// TIA Portal V20 export
DATA_BLOCK "BK05"   // DB194
// stored: MemoryReserve 100
   VAR
      "X10-1 SPARE" : Bool;
      "X11-1 SPARE" : Bool;
      "X12-1 COMPENSATOR LIMIT SENSOR(-)" : Bool;
      "X13-1 COMPENSATOR LIMIT SENSOR(+)" : Bool;
      "X14-1 FEEDER CYLINDER UP" : Bool;
      "X15-1 VISION PUSHER SUPPORT UP" : Bool;
      "X16-1 ELECTRODE NG BOX LOCK CYLINDER DOWN" : Bool;
      "X17-1 UNWINDER DANCER SAFETY PIN IDLE POSITION" : Bool;
      "X10-2 SPARE" : Bool;
      "X11-2 SPARE" : Bool;
      "X12-2 COMPENSATOR HOMING SENSOR" : Bool;
      "X13-2 COMPENSATOR SAFETY PIN IDLE POSITION" : Bool;
      "X14-2 FEEDER CYLINDER DOWN" : Bool;
      "X15-2 VISION PUSHER SUPPORT DOWN" : Bool;
      "X16-2 ELECTRODE NG BOX LOCK CYLINDER UP" : Bool;
      "X17-2 SPARE" : Bool;
   END_VAR
BEGIN
END_DATA_BLOCK
